(* IEC 61131-3 sources: ArfBotOS/Codesys-4/ArfBotOS.fbsdev/Application.iecapp^/FUN/logic, 5 files *)

(* ---- F_BuildLogicCmd.fn.st ---- *)
FUNCTION F_BuildLogicCmd : STRING(GVL_App.COMMAND_LEN)
VAR_INPUT
	stCommand: ST_LogicCmd;
END_VAR
VAR
    _Command: STRING(GVL_App.COMMAND_LEN);
END_VAR
VAR CONSTANT
	_Delimiter: STRING:=' ';
END_VAR

// IF PASS|INPUT|REGISTER|COUNTER <index> >|<|=|>=|<= <value>
// THEN OUTPUT|JUMP|CNTUP|CNTDN|CNTRST|REGISTER|NOP <index> <value>
// ELSE OUTPUT|JUMP|CNTUP|CNTDN|CNTRST|REGISTER|NOP <index> <value>
//
// IF_Condition
// IF_Condition_Idx
// IF_Condition_Operator
// IF_Condition_Operator_Compare
// THEN_Function
// THEN_Function_Value
// THEN_Function_Idx
// ELSE_Function
// ELSE_Function_Idx
// ELSE_Function_Value

// clear the command
_Command:='';

// build command
F_AddElement(_Command, _Delimiter, 'IF');
F_AddElement(_Command, _Delimiter, TO_STRING(stCommand.IF_Condition));
IF stCommand.IF_Condition <> E_LogicIfCondition.PASS THEN
	F_AddElement(_Command, _Delimiter, INT_TO_STRING(stCommand.IF_Condition_Idx));
	F_AddElement(_Command, _Delimiter, TO_STRING(stCommand.IF_Condition_Operator));
	F_AddElement(_Command, _Delimiter, UDINT_TO_STRING(stCommand.IF_Condition_Operator_Value));
END_IF
F_AddElement(_Command, _Delimiter, 'THEN');
F_AddElement(_Command, _Delimiter, TO_STRING(stCommand.THEN_Function));
IF stCommand.THEN_Function <> E_LogicFunction.NOP THEN
	F_AddElement(_Command, _Delimiter, INT_TO_STRING(stCommand.THEN_Function_Idx));
	IF stCommand.THEN_Function = E_LogicFunction.OUTPUT OR
		stCommand.THEN_Function = E_LogicFunction.REGISTER OR
		stCommand.THEN_Function = E_LogicFunction.FLAG THEN
			F_AddElement(_Command, _Delimiter, UDINT_TO_STRING(stCommand.THEN_Function_Value));
	END_IF
END_IF
IF stCommand.IF_Condition <> E_LogicIfCondition.PASS THEN
	F_AddElement(_Command, _Delimiter, 'ELSE');
	F_AddElement(_Command, _Delimiter, TO_STRING(stCommand.ELSE_Function));
	IF stCommand.ELSE_Function <> E_LogicFunction.NOP THEN
		F_AddElement(_Command, _Delimiter, INT_TO_STRING(stCommand.ELSE_Function_Idx));
		IF stCommand.ELSE_Function = E_LogicFunction.OUTPUT OR
			stCommand.ELSE_Function = E_LogicFunction.REGISTER OR
			stCommand.ELSE_Function = E_LogicFunction.FLAG THEN
				F_AddElement(_Command, _Delimiter, UDINT_TO_STRING(stCommand.ELSE_Function_Value));
		END_IF
	END_IF
END_IF

// set function equal to command
F_BuildLogicCmd := _Command;
END_FUNCTION

(* ---- F_ChangeJumpRow.fn.st ---- *)
FUNCTION F_ChangeJumpRow : BOOL
VAR_IN_OUT
	Command: DUT_Command;
END_VAR
VAR_INPUT
	BeginningRow: DINT;
	Change: INT;
END_VAR
VAR
	_LogicCmdParser : FB_ParseLogicCmd;
	_stLogicCmd : ST_LogicCmd;
END_VAR

// change the row that the jump function will jump to by the amount of the change
F_ChangeJumpRow := FALSE;
IF Command.CommandType = DUT_CommandType.LogicCommand THEN
	// parse the command string
	_LogicCmdParser(Command:=Command.CommandString, stCommand=>_stLogicCmd);

	// check the THEN function
	IF _stLogicCmd.THEN_Function = E_LogicFunction.JUMP AND_THEN _stLogicCmd.THEN_Function_Idx >= BeginningRow THEN
		_stLogicCmd.THEN_Function_Idx := _stLogicCmd.THEN_Function_Idx + Change;
		F_ChangeJumpRow := TRUE;
	END_IF

	// check the ELSE function
	IF _stLogicCmd.ELSE_Function = E_LogicFunction.JUMP AND_THEN _stLogicCmd.ELSE_Function_Idx >= BeginningRow  THEN
		_stLogicCmd.ELSE_Function_Idx := _stLogicCmd.ELSE_Function_Idx + Change;
		F_ChangeJumpRow := TRUE;
	END_IF

	// set the command
	IF F_ChangeJumpRow THEN
		Command.CommandString := F_BuildLogicCmd(stCommand:=_stLogicCmd);
	END_IF

ELSE
	F_ChangeJumpRow := FALSE;

END_IF
END_FUNCTION

(* ---- F_SplitCmd.fn.st ---- *)
FUNCTION F_SplitCmd : ARRAY [0..GVL_App.COMMAND_LEN] OF STRING
VAR_INPUT
    Command: STRING(GVL_App.COMMAND_LEN);
	Delimiter: STRING(1):=' ';
END_VAR
VAR
	_Command: STRING(GVL_App.COMMAND_LEN);
	_DelimPos: INT;
	_i, _j, _k: INT;
END_VAR
VAR CONSTANT
	_SpaceChar: STRING(1):=' ';
END_VAR

// grab a copy
// TODO do we need to do this? cant we just operate on the input?
_Command := Command;

// ex. 123 456 789 0 123 456 879 0
WHILE LEN(_Command) > 0  AND _i < GVL_App.COMMAND_LEN DO
	// find the delimiter
	_DelimPos := FIND(_Command, Delimiter);
	// don't copy empty commands
	IF _DelimPos > 1 THEN
		// copy the command into the array position
		F_SplitCmd[_i] := MID(STR:=_Command, LEN:=_DelimPos - 1, POS:=1);
		// trim the command off the front of the string
		_Command := DELETE(STR:=_Command, LEN:=_DelimPos, POS:=1);
		// increment the index and get ready for the next
		_i := _i + 1;
	ELSIF _DelimPos = 1 OR FIND(_Command, _SpaceChar) = 1 THEN
		// don't do anything with a stray delimiter or a space at the  start of the next command
		// trim the command off the space at the front of the string
		_Command := DELETE(STR:=_Command, LEN:=LEN(_SpaceChar), POS:=1);
	ELSIF _DelimPos = 0 AND LEN(_Command) > 0 THEN
		// copy the last command into the array position and return
		F_SplitCmd[_i] := MID(STR:=_Command, LEN:=LEN(_Command), POS:=1);
		// trim the command off the front of the string
		_Command := DELETE(STR:=_Command, LEN:=_DelimPos, POS:=1);
		// increment the index and get ready for the next
		_i := _i + 1;
		RETURN;
	ELSE
		RETURN;
	END_IF
END_WHILE
END_FUNCTION

(* ---- FB_LogicCmdProcessor.fb.st ---- *)
FUNCTION_BLOCK FB_LogicCmdProcessor EXTENDS FB_Module
VAR_IN_OUT
	PrgProcessor: FB_ProgramProcessor;
	CmdProcessor: FB_CommandProcessor;
	CmdIO: ST_LogicCmdIO;
END_VAR
VAR_INPUT
	Command: STRING(GVL_App.COMMAND_LEN):='';
END_VAR
VAR_OUTPUT
END_VAR
VAR
	_UnitModeCurrentState: PACK_ML.State;
	_ParseLogicCmd: FB_ParseLogicCmd;
	_ThenFunctionProcessed: BOOL;
END_VAR
VAR CONSTANT
	_STEP_DONE: 		INT := 1000;
	_STEP_IDLE: 		INT := 0000;
	_STEP_COMMAND: 		INT := 0010;
	_STEP_ERR: 			INT := 0020;
	_STEP_EVAL_IN:		INT := 0100;
	_STEP_EVAL_REG:		INT := 0110;
	_STEP_EVAL_CNT:		INT := 0120;
	_STEP_PROC_THEN:	INT := 0200;
	_STEP_PROC_ELSE:	INT := 0210;
	_STEP_PROC_OUT:		INT := 0300;
	_STEP_PROC_JMP:		INT := 0310;
	_STEP_PROC_CNT:		INT := 0320;
	_STEP_PROC_FLG:		INT := 0325;
	_STEP_PROC_REG:		INT := 0330;
	_STEP_EVAL_FLG:		INT := 0335;
	_STEP_PROC_NOP:		INT := 0340;
	_STEP_PROC_CAL:		INT := 0350;
END_VAR

SUPER^();

// PackML state machine implementation
_UnitModeCurrentState := SUPER^._UnitMode.CurrentState;

//
CASE SUPER^._SeqMain OF

    _STEP_DONE:
		SUPER^._SeqMain := _STEP_IDLE;

    _STEP_IDLE:
		// wait here until commanded to start

    _STEP_COMMAND:
		_ParseLogicCmd(Command:=Command);

		CASE _ParseLogicCmd.stCommand.IF_Condition OF
			E_LogicIfCondition.PASS:
				SUPER^._SeqMain := _STEP_PROC_THEN;
			E_LogicIfCondition.INPUT:
				SUPER^._SeqMain := _STEP_EVAL_IN;
			E_LogicIfCondition.REGISTER:
				SUPER^._SeqMain := _STEP_EVAL_REG;
			E_LogicIfCondition.COUNTER:
				SUPER^._SeqMain := _STEP_EVAL_CNT;
			E_LogicIfCondition.FLAG:
				SUPER^._SeqMain := _STEP_EVAL_FLG;
		END_CASE

		//
		_ThenFunctionProcessed := FALSE;

	_STEP_EVAL_IN:
		CASE _ParseLogicCmd.stCommand.IF_Condition_Operator OF
			E_LogicIfConditionOperator.EQU:
				IF CmdIO.Input[_ParseLogicCmd.stCommand.IF_Condition_Idx]
					= UDINT_TO_BOOL(_ParseLogicCmd.stCommand.IF_Condition_Operator_Value) THEN
						SUPER^._SeqMain := _STEP_PROC_THEN;
				ELSE
					SUPER^._SeqMain := _STEP_PROC_ELSE;
				END_IF
			E_LogicIfConditionOperator.GRE:
				IF CmdIO.Input[_ParseLogicCmd.stCommand.IF_Condition_Idx]
					>= UDINT_TO_BOOL(_ParseLogicCmd.stCommand.IF_Condition_Operator_Value) THEN
						SUPER^._SeqMain := _STEP_PROC_THEN;
				ELSE
					SUPER^._SeqMain := _STEP_PROC_ELSE;
				END_IF
			E_LogicIfConditionOperator.GRT:
				IF CmdIO.Input[_ParseLogicCmd.stCommand.IF_Condition_Idx]
					> UDINT_TO_BOOL(_ParseLogicCmd.stCommand.IF_Condition_Operator_Value) THEN
						SUPER^._SeqMain := _STEP_PROC_THEN;
				ELSE
					SUPER^._SeqMain := _STEP_PROC_ELSE;
				END_IF
			E_LogicIfConditionOperator.LEQ:
				IF CmdIO.Input[_ParseLogicCmd.stCommand.IF_Condition_Idx]
					<= UDINT_TO_BOOL(_ParseLogicCmd.stCommand.IF_Condition_Operator_Value) THEN
						SUPER^._SeqMain := _STEP_PROC_THEN;
				ELSE
					SUPER^._SeqMain := _STEP_PROC_ELSE;
				END_IF
			E_LogicIfConditionOperator.LES:
				IF CmdIO.Input[_ParseLogicCmd.stCommand.IF_Condition_Idx]
					< UDINT_TO_BOOL(_ParseLogicCmd.stCommand.IF_Condition_Operator_Value) THEN
						SUPER^._SeqMain := _STEP_PROC_THEN;
				ELSE
					SUPER^._SeqMain := _STEP_PROC_ELSE;
				END_IF
		END_CASE

	_STEP_EVAL_REG:
		CASE _ParseLogicCmd.stCommand.IF_Condition_Operator OF
			E_LogicIfConditionOperator.EQU:
				IF CmdIO.Register[_ParseLogicCmd.stCommand.IF_Condition_Idx]
					= _ParseLogicCmd.stCommand.IF_Condition_Operator_Value THEN
						SUPER^._SeqMain := _STEP_PROC_THEN;
				ELSE
					SUPER^._SeqMain := _STEP_PROC_ELSE;
				END_IF
			E_LogicIfConditionOperator.GRE:
				IF CmdIO.Register[_ParseLogicCmd.stCommand.IF_Condition_Idx]
					>= _ParseLogicCmd.stCommand.IF_Condition_Operator_Value THEN
						SUPER^._SeqMain := _STEP_PROC_THEN;
				ELSE
					SUPER^._SeqMain := _STEP_PROC_ELSE;
				END_IF
			E_LogicIfConditionOperator.GRT:
				IF CmdIO.Register[_ParseLogicCmd.stCommand.IF_Condition_Idx]
					> _ParseLogicCmd.stCommand.IF_Condition_Operator_Value THEN
						SUPER^._SeqMain := _STEP_PROC_THEN;
				ELSE
					SUPER^._SeqMain := _STEP_PROC_ELSE;
				END_IF
			E_LogicIfConditionOperator.LEQ:
				IF CmdIO.Register[_ParseLogicCmd.stCommand.IF_Condition_Idx]
					<= _ParseLogicCmd.stCommand.IF_Condition_Operator_Value THEN
						SUPER^._SeqMain := _STEP_PROC_THEN;
				ELSE
					SUPER^._SeqMain := _STEP_PROC_ELSE;
				END_IF
			E_LogicIfConditionOperator.LES:
				IF CmdIO.Register[_ParseLogicCmd.stCommand.IF_Condition_Idx]
					< _ParseLogicCmd.stCommand.IF_Condition_Operator_Value THEN
						SUPER^._SeqMain := _STEP_PROC_THEN;
				ELSE
					SUPER^._SeqMain := _STEP_PROC_ELSE;
				END_IF
		END_CASE

	_STEP_EVAL_CNT:
		CASE _ParseLogicCmd.stCommand.IF_Condition_Operator OF
			E_LogicIfConditionOperator.EQU:
				IF CmdIO.Counter[_ParseLogicCmd.stCommand.IF_Condition_Idx]
					= _ParseLogicCmd.stCommand.IF_Condition_Operator_Value THEN
						SUPER^._SeqMain := _STEP_PROC_THEN;
				ELSE
					SUPER^._SeqMain := _STEP_PROC_ELSE;
				END_IF
			E_LogicIfConditionOperator.GRE:
				IF CmdIO.Counter[_ParseLogicCmd.stCommand.IF_Condition_Idx]
					>= _ParseLogicCmd.stCommand.IF_Condition_Operator_Value THEN
						SUPER^._SeqMain := _STEP_PROC_THEN;
				ELSE
					SUPER^._SeqMain := _STEP_PROC_ELSE;
				END_IF
			E_LogicIfConditionOperator.GRT:
				IF CmdIO.Counter[_ParseLogicCmd.stCommand.IF_Condition_Idx]
					> _ParseLogicCmd.stCommand.IF_Condition_Operator_Value THEN
						SUPER^._SeqMain := _STEP_PROC_THEN;
				ELSE
					SUPER^._SeqMain := _STEP_PROC_ELSE;
				END_IF
			E_LogicIfConditionOperator.LEQ:
				IF CmdIO.Counter[_ParseLogicCmd.stCommand.IF_Condition_Idx]
					<= _ParseLogicCmd.stCommand.IF_Condition_Operator_Value THEN
						SUPER^._SeqMain := _STEP_PROC_THEN;
				ELSE
					SUPER^._SeqMain := _STEP_PROC_ELSE;
				END_IF
			E_LogicIfConditionOperator.LES:
				IF CmdIO.Counter[_ParseLogicCmd.stCommand.IF_Condition_Idx]
					< _ParseLogicCmd.stCommand.IF_Condition_Operator_Value THEN
						SUPER^._SeqMain := _STEP_PROC_THEN;
				ELSE
					SUPER^._SeqMain := _STEP_PROC_ELSE;
				END_IF
		END_CASE

	_STEP_EVAL_FLG:
		CASE _ParseLogicCmd.stCommand.IF_Condition_Operator OF
			E_LogicIfConditionOperator.EQU:
				IF SUPER^.Flags[_ParseLogicCmd.stCommand.IF_Condition_Idx].Value
					= UDINT_TO_BOOL(_ParseLogicCmd.stCommand.IF_Condition_Operator_Value) THEN
						SUPER^._SeqMain := _STEP_PROC_THEN;
				ELSE
					SUPER^._SeqMain := _STEP_PROC_ELSE;
				END_IF
			E_LogicIfConditionOperator.GRE:
				IF SUPER^.Flags[_ParseLogicCmd.stCommand.IF_Condition_Idx].Value
					>= UDINT_TO_BOOL(_ParseLogicCmd.stCommand.IF_Condition_Operator_Value) THEN
						SUPER^._SeqMain := _STEP_PROC_THEN;
				ELSE
					SUPER^._SeqMain := _STEP_PROC_ELSE;
				END_IF
			E_LogicIfConditionOperator.GRT:
				IF SUPER^.Flags[_ParseLogicCmd.stCommand.IF_Condition_Idx].Value
					> UDINT_TO_BOOL(_ParseLogicCmd.stCommand.IF_Condition_Operator_Value) THEN
						SUPER^._SeqMain := _STEP_PROC_THEN;
				ELSE
					SUPER^._SeqMain := _STEP_PROC_ELSE;
				END_IF
			E_LogicIfConditionOperator.LEQ:
				IF SUPER^.Flags[_ParseLogicCmd.stCommand.IF_Condition_Idx].Value
					<= UDINT_TO_BOOL(_ParseLogicCmd.stCommand.IF_Condition_Operator_Value) THEN
						SUPER^._SeqMain := _STEP_PROC_THEN;
				ELSE
					SUPER^._SeqMain := _STEP_PROC_ELSE;
				END_IF
			E_LogicIfConditionOperator.LES:
				IF SUPER^.Flags[_ParseLogicCmd.stCommand.IF_Condition_Idx].Value
					< UDINT_TO_BOOL(_ParseLogicCmd.stCommand.IF_Condition_Operator_Value) THEN
						SUPER^._SeqMain := _STEP_PROC_THEN;
				ELSE
					SUPER^._SeqMain := _STEP_PROC_ELSE;
				END_IF
		END_CASE

	_STEP_PROC_THEN:
		//
		_ThenFunctionProcessed := TRUE;
		//
		CASE _ParseLogicCmd.stCommand.THEN_Function OF
			E_LogicFunction.OUTPUT:
				SUPER^._SeqMain := _STEP_PROC_OUT;
			E_LogicFunction.REGISTER:
				SUPER^._SeqMain := _STEP_PROC_REG;
			E_LogicFunction.FLAG:
				SUPER^._SeqMain := _STEP_PROC_FLG;
			E_LogicFunction.CNTUP:
				SUPER^._SeqMain := _STEP_PROC_CNT;
			E_LogicFunction.CNTDN:
				SUPER^._SeqMain := _STEP_PROC_CNT;
			E_LogicFunction.CNTRST:
				SUPER^._SeqMain := _STEP_PROC_CNT;
			E_LogicFunction.JUMP:
				SUPER^._SeqMain := _STEP_PROC_JMP;
			E_LogicFunction.CALL:
				SUPER^._SeqMain := _STEP_PROC_CAL;
			E_LogicFunction.NOP:
				SUPER^._SeqMain := _STEP_PROC_NOP;
		END_CASE;

	_STEP_PROC_ELSE:
		IF _ParseLogicCmd.stCommand.IF_Condition <> E_LogicIfCondition.PASS THEN
			CASE _ParseLogicCmd.stCommand.ELSE_Function OF
				E_LogicFunction.OUTPUT:
					SUPER^._SeqMain := _STEP_PROC_OUT;
				E_LogicFunction.REGISTER:
					SUPER^._SeqMain := _STEP_PROC_REG;
				E_LogicFunction.FLAG:
					SUPER^._SeqMain := _STEP_PROC_FLG;
				E_LogicFunction.CNTUP:
					SUPER^._SeqMain := _STEP_PROC_CNT;
				E_LogicFunction.CNTDN:
					SUPER^._SeqMain := _STEP_PROC_CNT;
				E_LogicFunction.CNTRST:
					SUPER^._SeqMain := _STEP_PROC_CNT;
				E_LogicFunction.JUMP:
					SUPER^._SeqMain := _STEP_PROC_JMP;
				E_LogicFunction.CALL:
					SUPER^._SeqMain := _STEP_PROC_CAL;
				E_LogicFunction.NOP:
					SUPER^._SeqMain := _STEP_PROC_NOP;
			END_CASE;
		ELSE
			SUPER^._SeqMain := _STEP_DONE;
		END_IF

	_STEP_PROC_OUT:
		IF _ThenFunctionProcessed THEN
			CmdIO.Output[_ParseLogicCmd.stCommand.THEN_Function_Idx]
				:= UDINT_TO_BOOL(_ParseLogicCmd.stCommand.THEN_Function_Value);
		ELSE
			CmdIO.Output[_ParseLogicCmd.stCommand.ELSE_Function_Idx]
				:= UDINT_TO_BOOL(_ParseLogicCmd.stCommand.ELSE_Function_Value);
		END_IF
		// next, please
		SUPER^._SeqMain := _STEP_DONE;

	_STEP_PROC_REG:
		IF _ThenFunctionProcessed THEN
			CmdIO.Register[_ParseLogicCmd.stCommand.THEN_Function_Idx]
				:= _ParseLogicCmd.stCommand.THEN_Function_Value;
		ELSE
			CmdIO.Register[_ParseLogicCmd.stCommand.ELSE_Function_Idx]
				:= _ParseLogicCmd.stCommand.ELSE_Function_Value;
		END_IF
		// next, please
		SUPER^._SeqMain := _STEP_DONE;

	_STEP_PROC_CNT:
		IF _ThenFunctionProcessed THEN
			CASE _ParseLogicCmd.stCommand.THEN_Function OF
				E_LogicFunction.CNTUP:
					CmdIO.Counter[_ParseLogicCmd.stCommand.THEN_Function_Idx]
						:= CmdIO.Counter[_ParseLogicCmd.stCommand.THEN_Function_Idx] + 1;
				E_LogicFunction.CNTDN:
					CmdIO.Counter[_ParseLogicCmd.stCommand.THEN_Function_Idx]
						:= CmdIO.Counter[_ParseLogicCmd.stCommand.THEN_Function_Idx] - 1;
				E_LogicFunction.CNTRST:
					CmdIO.Counter[_ParseLogicCmd.stCommand.THEN_Function_Idx]
						:= 0;
			END_CASE
		ELSE
			CASE _ParseLogicCmd.stCommand.ELSE_Function OF
				E_LogicFunction.CNTUP:
					CmdIO.Counter[_ParseLogicCmd.stCommand.ELSE_Function_Idx]
						:= CmdIO.Counter[_ParseLogicCmd.stCommand.ELSE_Function_Idx] + 1;
				E_LogicFunction.CNTDN:
					CmdIO.Counter[_ParseLogicCmd.stCommand.ELSE_Function_Idx]
						:= CmdIO.Counter[_ParseLogicCmd.stCommand.ELSE_Function_Idx] - 1;
				E_LogicFunction.CNTRST:
					CmdIO.Counter[_ParseLogicCmd.stCommand.ELSE_Function_Idx]
						:= 0;
			END_CASE
		END_IF
		// next, please
		SUPER^._SeqMain := _STEP_DONE;

	_STEP_PROC_FLG:
		IF _ThenFunctionProcessed THEN
			SUPER^.Flags[_ParseLogicCmd.stCommand.THEN_Function_Idx].Value
				:= UDINT_TO_BOOL(_ParseLogicCmd.stCommand.THEN_Function_Value);
		ELSE
			SUPER^.Flags[_ParseLogicCmd.stCommand.ELSE_Function_Idx].Value
				:= UDINT_TO_BOOL(_ParseLogicCmd.stCommand.ELSE_Function_Value);
		END_IF
		// next, please
		SUPER^._SeqMain := _STEP_DONE;

	_STEP_PROC_JMP:
		IF _ThenFunctionProcessed THEN
			CmdProcessor.M_SetNextCommand(CommandNumber:=INT_TO_UINT(_ParseLogicCmd.stCommand.THEN_Function_Idx));
		ELSE
			CmdProcessor.M_SetNextCommand(CommandNumber:=INT_TO_UINT(_ParseLogicCmd.stCommand.ELSE_Function_Idx));
		END_IF
		// next, please
		SUPER^._SeqMain := _STEP_DONE;

	_STEP_PROC_CAL:
		IF _ThenFunctionProcessed THEN
			PrgProcessor.M_CallProgram(	ProgramNumber:= INT_TO_UINT(_ParseLogicCmd.stCommand.THEN_Function_Idx),
										ReturnProgram:= PrgProcessor.P_CurrentProgram,
										ReturnCommand:= CmdProcessor.P_CurrentCommandIndex);
		ELSE
			PrgProcessor.M_CallProgram(	ProgramNumber:= INT_TO_UINT(_ParseLogicCmd.stCommand.ELSE_Function_Idx),
										ReturnProgram:= PrgProcessor.P_CurrentProgram,
										ReturnCommand:= CmdProcessor.P_CurrentCommandIndex);
		END_IF
		// next, please
		SUPER^._SeqMain := _STEP_DONE;

	_STEP_PROC_NOP:
		IF _ThenFunctionProcessed THEN
			//
		ELSE
			//
		END_IF
		// next, please
		SUPER^._SeqMain := _STEP_DONE;

END_CASE
END_FUNCTION_BLOCK

(* ---- FB_ParseLogicCmd.fb.st ---- *)
FUNCTION_BLOCK FB_ParseLogicCmd
VAR_INPUT
	Command: STRING(GVL_App.COMMAND_LEN);
END_VAR
VAR_OUTPUT
	stCommand: ST_LogicCmd;
	Error: BOOL;
	ErrorDescription: STRING;
END_VAR
VAR
	_CmdParams: ARRAY [0..GVL_App.COMMAND_LEN] OF STRING;
	_i, _j, _k: INT;
END_VAR

// IF PASS|INPUT|REGISTER|COUNTER <index> >|<|=|>=|<= <value>
// THEN OUTPUT|JUMP|CALL|CNTUP|CNTDN|CNTRST|REGISTER|NOP <index> <value>
// ELSE OUTPUT|JUMP|CALL|CNTUP|CNTDN|CNTRST|REGISTER|NOP <index> <value>
//
// IF_Condition
// IF_Condition_Idx
// IF_Condition_Operator
// IF_Condition_Operator_Compare
// THEN_Function
// THEN_Function_Value
// THEN_Function_Idx
// ELSE_Function
// ELSE_Function_Idx
// ELSE_Function_Value

Error:=FALSE;
ErrorDescription:='';

// split command string into commands
_CmdParams:=F_SplitCmd(Command:=Command);

//
_i := 0;

// disregard the 'IF'
_i := _i + 1;

//
IF _CmdParams[_i] = TO_STRING(E_LogicIfCondition.PASS) THEN
	stCommand.IF_Condition := E_LogicIfCondition.PASS;
ELSIF  _CmdParams[_i] = TO_STRING(E_LogicIfCondition.INPUT) THEN
	stCommand.IF_Condition := E_LogicIfCondition.INPUT;
ELSIF  _CmdParams[_i] = TO_STRING(E_LogicIfCondition.REGISTER) THEN
	stCommand.IF_Condition := E_LogicIfCondition.REGISTER;
ELSIF  _CmdParams[_i] = TO_STRING(E_LogicIfCondition.COUNTER) THEN
	stCommand.IF_Condition := E_LogicIfCondition.COUNTER;
ELSIF  _CmdParams[_i] = TO_STRING(E_LogicIfCondition.FLAG) THEN
	stCommand.IF_Condition := E_LogicIfCondition.FLAG;
END_IF
_i := _i + 1;

//
IF stCommand.IF_Condition <> E_LogicIfCondition.PASS THEN

	//
	stCommand.IF_Condition_Idx := STRING_TO_INT(_CmdParams[_i]);
	_i := _i + 1;

	//
	IF _CmdParams[_i] = TO_STRING(E_LogicIfConditionOperator.GRT) THEN
		stCommand.IF_Condition_Operator := E_LogicIfConditionOperator.GRT;
	ELSIF _CmdParams[_i] = TO_STRING(E_LogicIfConditionOperator.LES) THEN
		stCommand.IF_Condition_Operator := E_LogicIfConditionOperator.LES;
	ELSIF _CmdParams[_i] = TO_STRING(E_LogicIfConditionOperator.EQU) THEN
		stCommand.IF_Condition_Operator := E_LogicIfConditionOperator.EQU;
	ELSIF _CmdParams[_i] = TO_STRING(E_LogicIfConditionOperator.GRE) THEN
		stCommand.IF_Condition_Operator := E_LogicIfConditionOperator.GRE;
	ELSIF _CmdParams[_i] = TO_STRING(E_LogicIfConditionOperator.LEQ) THEN
		stCommand.IF_Condition_Operator := E_LogicIfConditionOperator.LEQ;
	END_IF
	_i := _i + 1;

	//
	stCommand.IF_Condition_Operator_Value := STRING_TO_UDINT(_CmdParams[_i]);
	_i := _i + 1;

END_IF

// disregard the 'THEN'
_i := _i + 1;

//
IF _CmdParams[_i] = TO_STRING(E_LogicFunction.OUTPUT) THEN
	stCommand.THEN_Function := E_LogicFunction.OUTPUT;
ELSIF _CmdParams[_i] = TO_STRING(E_LogicFunction.JUMP) THEN
	stCommand.THEN_Function := E_LogicFunction.JUMP;
ELSIF _CmdParams[_i] = TO_STRING(E_LogicFunction.CALL) THEN
	stCommand.THEN_Function := E_LogicFunction.CALL;
ELSIF _CmdParams[_i] = TO_STRING(E_LogicFunction.CNTUP) THEN
	stCommand.THEN_Function := E_LogicFunction.CNTUP;
ELSIF _CmdParams[_i] = TO_STRING(E_LogicFunction.CNTDN) THEN
	stCommand.THEN_Function := E_LogicFunction.CNTDN;
ELSIF _CmdParams[_i] = TO_STRING(E_LogicFunction.CNTRST) THEN
	stCommand.THEN_Function := E_LogicFunction.CNTRST;
ELSIF _CmdParams[_i] = TO_STRING(E_LogicFunction.REGISTER) THEN
	stCommand.THEN_Function := E_LogicFunction.REGISTER;
ELSIF _CmdParams[_i] = TO_STRING(E_LogicFunction.FLAG) THEN
	stCommand.THEN_Function := E_LogicFunction.FLAG;
ELSIF _CmdParams[_i] = TO_STRING(E_LogicFunction.NOP) THEN
	stCommand.THEN_Function := E_LogicFunction.NOP;
END_IF
_i := _i + 1;

//
IF stCommand.THEN_Function <> E_LogicFunction.NOP THEN
	stCommand.THEN_Function_Idx := STRING_TO_INT(_CmdParams[_i]);
	_i := _i + 1;
	IF stCommand.THEN_Function = E_LogicFunction.OUTPUT OR
		stCommand.THEN_Function = E_LogicFunction.REGISTER OR
		stCommand.THEN_Function = E_LogicFunction.FLAG THEN
			stCommand.THEN_Function_Value := STRING_TO_UDINT(_CmdParams[_i]);
			_i := _i + 1;
	END_IF
END_IF

// disregard the 'ELSE'
_i := _i + 1;

//
IF _CmdParams[_i] = TO_STRING(E_LogicFunction.OUTPUT) THEN
	stCommand.ELSE_Function := E_LogicFunction.OUTPUT;
ELSIF _CmdParams[_i] = TO_STRING(E_LogicFunction.JUMP) THEN
	stCommand.ELSE_Function := E_LogicFunction.JUMP;
ELSIF _CmdParams[_i] = TO_STRING(E_LogicFunction.CALL) THEN
	stCommand.ELSE_Function := E_LogicFunction.CALL;
ELSIF _CmdParams[_i] = TO_STRING(E_LogicFunction.CNTUP) THEN
	stCommand.ELSE_Function := E_LogicFunction.CNTUP;
ELSIF _CmdParams[_i] = TO_STRING(E_LogicFunction.CNTDN) THEN
	stCommand.ELSE_Function := E_LogicFunction.CNTDN;
ELSIF _CmdParams[_i] = TO_STRING(E_LogicFunction.CNTRST) THEN
	stCommand.ELSE_Function := E_LogicFunction.CNTRST;
ELSIF _CmdParams[_i] = TO_STRING(E_LogicFunction.REGISTER) THEN
	stCommand.ELSE_Function := E_LogicFunction.REGISTER;
ELSIF _CmdParams[_i] = TO_STRING(E_LogicFunction.FLAG) THEN
	stCommand.ELSE_Function := E_LogicFunction.FLAG;
ELSIF _CmdParams[_i] = TO_STRING(E_LogicFunction.NOP) THEN
	stCommand.ELSE_Function := E_LogicFunction.NOP;
END_IF
_i := _i + 1;

//
IF stCommand.ELSE_Function <> E_LogicFunction.NOP THEN
	stCommand.ELSE_Function_Idx := STRING_TO_INT(_CmdParams[_i]);
	_i := _i + 1;
	IF stCommand.ELSE_Function = E_LogicFunction.OUTPUT OR
		stCommand.ELSE_Function = E_LogicFunction.REGISTER OR
		stCommand.ELSE_Function = E_LogicFunction.FLAG THEN
			stCommand.ELSE_Function_Value := STRING_TO_UDINT(_CmdParams[_i]);
			_i := _i + 1;
	END_IF
END_IF
END_FUNCTION_BLOCK
